program PRG_Syntax_Main  
var  
    _nCycle : udint;  
    _bReady       : bool;  
end_var

_nCycle := _nCycle + 1;
_bReady := true;

END_PROGRAM

(* stored: Version 1.1.0.1, ProductVersion 3.1.4024.16
   POU PRG_Syntax_Main: Id {c1891f57-0da9-4e5c-b324-15acd7b61c68}, SpecialFunc None *)
